PROGRAM MAIN
VAR
END_VAR

AutomationLibrary();
Visualaisation_Control();
RobotPosTracker();

Robot();
AutoMode();
ModeControl();
ManualMode();

END_PROGRAM

(* stored: Version 1.1.0.1, ProductVersion 3.1.4024.12
   POU MAIN: Id {eedc87b0-498f-42a3-9add-b62d0d4a527c}, SpecialFunc None *)
